// TIA Portal V20 export
TYPE "LBP_typeInternal5"
TITLE = Internal data type for basic program / Type de données interne pour programme de base
// Data type only for internal use in the basic program / Type de données réservé à l'utilisation interne dans le programme de base
   STRUCT
      accepted : Bool;
      abort : Bool;
      writeRecord : Bool;
      mcpNumber : UInt;
      slotNumber : UInt;
      recordNumber : UInt;
      recordLength : UInt;
      recordData : Array[0..223] of Byte;
      done : Bool;
      busy : Bool;
      error : Bool;
      status : Word;
   END_STRUCT;
END_TYPE
